FUNCTION_BLOCK Recipe_10054_Sixteen
VAR_INPUT
	execute: BOOL;
	Order: DUT_RECIPEORDER;
END_VAR
VAR_OUTPUT
	RecipeInfo: DUT_RECIPEOFFER;
	RecipeDone: BOOL;
	InitDone: BOOL;
	Ready: BOOL;
END_VAR
VAR
	userparametersum: LREAL;
	StepDone: BOOL;
	i: INT;
	Command: ARRAY[1..5] OF DUT_RecipeCommand;
	NextSkill: BOOL;
	SectionReady: BOOL;
END_VAR

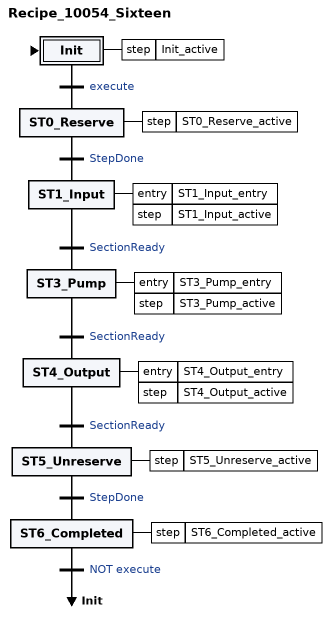
INITIAL_STEP Init:
    Init_active(N);  // step action
END_STEP
TRANSITION FROM Init TO ST0_Reserve
    := execute;
END_TRANSITION
STEP ST0_Reserve:
    ST0_Reserve_active(N);  // step action
END_STEP
TRANSITION FROM ST0_Reserve TO ST1_Input
    := StepDone;
END_TRANSITION
STEP ST1_Input:
    ST1_Input_entry(P1);  // entry action
    ST1_Input_active(N);  // step action
END_STEP
TRANSITION FROM ST1_Input TO ST3_Pump
    := SectionReady;
END_TRANSITION
STEP ST3_Pump:
    ST3_Pump_entry(P1);  // entry action
    ST3_Pump_active(N);  // step action
END_STEP
TRANSITION FROM ST3_Pump TO ST4_Output
    := SectionReady;
END_TRANSITION
STEP ST4_Output:
    ST4_Output_entry(P1);  // entry action
    ST4_Output_active(N);  // step action
END_STEP
TRANSITION FROM ST4_Output TO ST5_Unreserve
    := SectionReady;
END_TRANSITION
STEP ST5_Unreserve:
    ST5_Unreserve_active(N);  // step action
END_STEP
TRANSITION FROM ST5_Unreserve TO ST6_Completed
    := StepDone;
END_TRANSITION
STEP ST6_Completed:
    ST6_Completed_active(N);  // step action
END_STEP
TRANSITION FROM ST6_Completed TO Init
    := NOT execute;
END_TRANSITION

ACTION ST32b_Dose_exit:

END_ACTION

ACTION ST40_TransOutput_active:
//RT: 2014.11.23: Mover zum Output
StepDone := FALSE;

//Skill auswählen
ExecuteSkill.SkillID 		:= 1320;
ExecuteSkill.SkillName	 	:= 'Transport';

//Parameter setzen

ExecuteSkill.Parameter[3].ID := 3;
ExecuteSkill.Parameter[3].Name := 'Velocity';
ExecuteSkill.Parameter[3].Value := 300;



ExecuteSkill.Parameter[1].ID :=  1;
ExecuteSkill.Parameter[1].Name := 'TargetPosition X';
ExecuteSkill.Parameter[1].Value := 30 ;
ExecuteSkill.Parameter[1].StringValue := '#DP#2#XPosition';



ExecuteSkill.Parameter[2].ID := 2;
ExecuteSkill.Parameter[2].Name := 'TargetPosition Z';
ExecuteSkill.Parameter[2].Value := 100;// ZCookieModule - ZCookieModuleCalibration - 2* Cookiethickness + toppingthickness+ Preasureheight  ;



(* ExecuteSkill.Parameter[4].ID := 4;
ExecuteSkill.Parameter[4].Name := 'Acceleration';
ExecuteSkill.Parameter[4].Value :=0 ;

*)
(*
ExecuteSkill.Parameter[5].ID := ;
ExecuteSkill.Parameter[5].Name := '';
ExecuteSkill.Parameter[5].Value := ;
*)



ExecuteSkill();

StepDone := ExecuteSkill.Done;
END_ACTION

ACTION ST12_Input_active:
//RT: 2014.11.23: Input Modul auslösen
StepDone := FALSE;

//Skill auswählen
ExecuteSkill.SkillID 		:= 1402;
ExecuteSkill.SkillName	 	:= 'Input';

//Parameter setzen

ExecuteSkill.Parameter[1].ID := 1;
ExecuteSkill.Parameter[1].Name := 'TaskID';
ExecuteSkill.Parameter[1].Value := Order.TaskID;


(*
ExecuteSkill.Parameter[2].ID := ;
ExecuteSkill.Parameter[2].Name := '';
ExecuteSkill.Parameter[2].Value := ;
*)

(*
ExecuteSkill.Parameter[3].ID := ;
ExecuteSkill.Parameter[3].Name := '';
ExecuteSkill.Parameter[3].Value := ;
*)

(*
ExecuteSkill.Parameter[4].ID := ;
ExecuteSkill.Parameter[4].Name := '';
ExecuteSkill.Parameter[4].Value := ;
*)

(*
ExecuteSkill.Parameter[5].ID := ;
ExecuteSkill.Parameter[5].Name := '';
ExecuteSkill.Parameter[5].Value := ;
*)



ExecuteSkill();

StepDone := ExecuteSkill.Done;
END_ACTION

ACTION ST13_UnblockInput_active:
//RT: 2014.11.23: Gibt Mover Position Frei
StepDone := FALSE;

//Skill auswählen
ExecuteSkill.SkillID 		:= 1316;
ExecuteSkill.SkillName	 	:= 'Unblock';

//Parameter setzen

ExecuteSkill.Parameter[1].ID := 1;
ExecuteSkill.Parameter[1].Name := 'TaskID';
ExecuteSkill.Parameter[1].Value := Order.TaskID;


(*
ExecuteSkill.Parameter[2].ID := ;
ExecuteSkill.Parameter[2].Name := '';
ExecuteSkill.Parameter[2].Value := ;
*)

(*
ExecuteSkill.Parameter[3].ID := ;
ExecuteSkill.Parameter[3].Name := '';
ExecuteSkill.Parameter[3].Value := ;
*)

(*
ExecuteSkill.Parameter[4].ID := ;
ExecuteSkill.Parameter[4].Name := '';
ExecuteSkill.Parameter[4].Value := ;
*)

(*
ExecuteSkill.Parameter[5].ID := ;
ExecuteSkill.Parameter[5].Name := '';
ExecuteSkill.Parameter[5].Value := ;
*)



ExecuteSkill();

StepDone := ExecuteSkill.Done;
END_ACTION

ACTION ST42_CocktailOutput_active:
//RT: 2014.11.23: Ausgeben des Produktes
StepDone := FALSE;

//Skill auswählen
ExecuteSkill.SkillID 		:= 1403;
ExecuteSkill.SkillName	 	:= 'Output';

//Parameter setzen

ExecuteSkill.Parameter[1].ID := 1;
ExecuteSkill.Parameter[1].Name := 'TaskID';
ExecuteSkill.Parameter[1].Value := Order.TaskID;


(*
ExecuteSkill.Parameter[2].ID := ;
ExecuteSkill.Parameter[2].Name := '';
ExecuteSkill.Parameter[2].Value := ;
*)

(*
ExecuteSkill.Parameter[3].ID := ;
ExecuteSkill.Parameter[3].Name := '';
ExecuteSkill.Parameter[3].Value := ;
*)

(*
ExecuteSkill.Parameter[4].ID := ;
ExecuteSkill.Parameter[4].Name := '';
ExecuteSkill.Parameter[4].Value := ;
*)

(*
ExecuteSkill.Parameter[5].ID := ;
ExecuteSkill.Parameter[5].Name := '';
ExecuteSkill.Parameter[5].Value := ;
*)



ExecuteSkill();

StepDone := ExecuteSkill.Done;
END_ACTION

ACTION ST6_Completed_active:
//RT: 2014.11.23: Warte auf Execute = False
RecipeDone := TRUE;
StepDone := FALSE;
END_ACTION

ACTION ST4_Output_entry:
SectionReady := FALSE;
END_ACTION

ACTION ST44_Exit_active:
SectionReady := TRUE;
END_ACTION

ACTION ST4_Output_active:
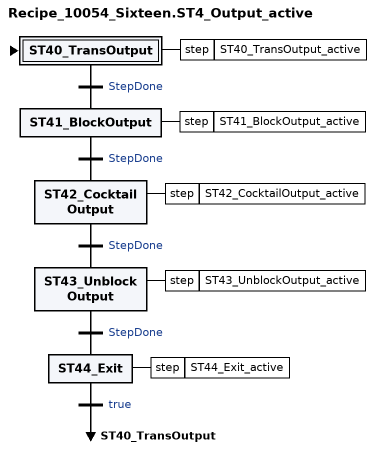
INITIAL_STEP ST40_TransOutput:
    ST40_TransOutput_active(N);  // step action
END_STEP
TRANSITION FROM ST40_TransOutput TO ST41_BlockOutput
    := StepDone;
END_TRANSITION
STEP ST41_BlockOutput:
    ST41_BlockOutput_active(N);  // step action
END_STEP
TRANSITION FROM ST41_BlockOutput TO ST42_CocktailOutput
    := StepDone;
END_TRANSITION
STEP ST42_CocktailOutput:
    ST42_CocktailOutput_active(N);  // step action
END_STEP
TRANSITION FROM ST42_CocktailOutput TO ST43_UnblockOutput
    := StepDone;
END_TRANSITION
STEP ST43_UnblockOutput:
    ST43_UnblockOutput_active(N);  // step action
END_STEP
TRANSITION FROM ST43_UnblockOutput TO ST44_Exit
    := StepDone;
END_TRANSITION
STEP ST44_Exit:
    ST44_Exit_active(N);  // step action
END_STEP
TRANSITION FROM ST44_Exit TO ST40_TransOutput
    := true;
END_TRANSITION
END_ACTION

ACTION Init_active:
//RT: 2014.11.23: Vorbereiten der daten und der HMI
RecipeDone := FALSE;

// Initialisation of Recipe Parameters an name etc
RecipeInfo.Name := 'Sixteen';
RecipeInfo.Description := '';
RecipeInfo.Dummy := FALSE;
RecipeInfo.RecipeID := 10054; 	// 
Initdone := TRUE;

//RT: 2014.11.23: wenn weniger als 5 alle lehren skills SkillID := 0
Command[1].SkillID := 1111;
Command[1].SkillName := 'Grenadine Syrup';
Command[1].Quantity := 11;

Command[2].SkillID := 1112;
Command[2].SkillName := 'Lemon Juice';
Command[2].Quantity := 11;

Command[3].SkillID := 1114;
Command[3].SkillName := 'Pineapple Juice';
Command[3].Quantity := 22;

Command[4].SkillID := 1117;
Command[4].SkillName := 'Orange Juice';
Command[4].Quantity := 45;

Command[5].SkillID := 1113;
Command[5].SkillName := 'Maracuja Juice';
Command[5].Quantity := 11;








//Parameter 0:

	RecipeInfo.UserParameter[0].Dummy 		:= FALSE;
	RecipeInfo.UserParameter[0].Default		:= 200;
	RecipeInfo.UserParameter[0].Description	:= 'Gives the total fluid amount in the glass';
	RecipeInfo.UserParameter[0].MaxValue	:= 200;
	RecipeInfo.UserParameter[0].MinValue	:= 10;
	RecipeInfo.UserParameter[0].Name		:= 'Total Liquid Amount';
	RecipeInfo.UserParameter[0].Unit		:= 'ml';
	
//Parameter 1-5:
FOR i := 1 TO 5 DO
	IF Command[i].SkillID = 0 THEN
		RecipeInfo.UserParameter[i].Dummy 		:= TRUE;
	ELSE
		RecipeInfo.UserParameter[i].Dummy 		:= FALSE;
		RecipeInfo.UserParameter[i].Default		:= Command[i].Quantity;
		RecipeInfo.UserParameter[i].Description	:= Command[i].SkillName;
		RecipeInfo.UserParameter[i].MaxValue	:= 100;
		RecipeInfo.UserParameter[i].MinValue	:= 1;
		RecipeInfo.UserParameter[i].Name		:= Command[i].SkillName;
		RecipeInfo.UserParameter[i].Unit		:= 'ml';	
	END_IF
END_FOR
END_ACTION

ACTION ST3_Pump_active:
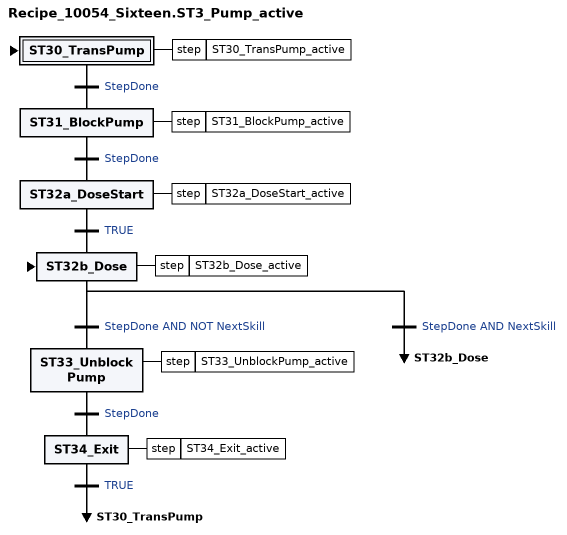
INITIAL_STEP ST30_TransPump:
    ST30_TransPump_active(N);  // step action
END_STEP
TRANSITION FROM ST30_TransPump TO ST31_BlockPump
    := StepDone;
END_TRANSITION
STEP ST31_BlockPump:
    ST31_BlockPump_active(N);  // step action
END_STEP
TRANSITION FROM ST31_BlockPump TO ST32a_DoseStart
    := StepDone;
END_TRANSITION
STEP ST32a_DoseStart:
    ST32a_DoseStart_active(N);  // step action
END_STEP
TRANSITION FROM ST32a_DoseStart TO ST32b_Dose
    := TRUE;
END_TRANSITION
STEP ST32b_Dose:
    ST32b_Dose_active(N);  // step action
END_STEP
TRANSITION FROM ST32b_Dose TO ST33_UnblockPump
    := StepDone AND NOT NextSkill;
END_TRANSITION
STEP ST33_UnblockPump:
    ST33_UnblockPump_active(N);  // step action
END_STEP
TRANSITION FROM ST33_UnblockPump TO ST34_Exit
    := StepDone;
END_TRANSITION
STEP ST34_Exit:
    ST34_Exit_active(N);  // step action
END_STEP
TRANSITION FROM ST34_Exit TO ST30_TransPump
    := TRUE;
END_TRANSITION
TRANSITION FROM ST32b_Dose TO ST32b_Dose
    := StepDone AND NextSkill;
END_TRANSITION
END_ACTION

ACTION ST34_Exit_active:
SectionReady := TRUE;
END_ACTION

ACTION ST10_TransToInput_active:
//RT: 2014.11.23: Mover zum Input

StepDone := FALSE;

//Skill auswählen
ExecuteSkill.SkillID 		:= 1320;
ExecuteSkill.SkillName	 	:= 'Transport';

//Parameter setzen

ExecuteSkill.Parameter[3].ID := 3;
ExecuteSkill.Parameter[3].Name := 'Velocity';
ExecuteSkill.Parameter[3].Value := 1000;



ExecuteSkill.Parameter[1].ID :=  1;
ExecuteSkill.Parameter[1].Name := 'TargetPosition X';
ExecuteSkill.Parameter[1].Value := 30 ;
ExecuteSkill.Parameter[1].StringValue := '#DP#2#XPosition';



ExecuteSkill.Parameter[2].ID := 2;
ExecuteSkill.Parameter[2].Name := 'TargetPosition Z';
ExecuteSkill.Parameter[2].Value := 100;// ZCookieModule - ZCookieModuleCalibration - 2* Cookiethickness + toppingthickness+ Preasureheight  ;



(*
ExecuteSkill.Parameter[4].ID := 4;
ExecuteSkill.Parameter[4].Name := 'Acceleration';
ExecuteSkill.Parameter[4].Value := 0 ;
*)

(*
ExecuteSkill.Parameter[5].ID := ;
ExecuteSkill.Parameter[5].Name := '';
ExecuteSkill.Parameter[5].Value := ;
*)



ExecuteSkill();

StepDone := ExecuteSkill.Done;
END_ACTION

ACTION ST1_Input_entry:
SectionReady := FALSE;
END_ACTION

ACTION ST32b_Dose_active:
//RT: 2014.11.23: Die Dosir Skills anlegen
StepDone := FALSE;

//Skill auswählen
ExecuteSkill.SkillID 		:= Command[i].SkillID;
ExecuteSkill.SkillName	 	:= Command[i].SkillName;
//Parameter setzen

ExecuteSkill.Parameter[0].ID := 1;
ExecuteSkill.Parameter[0].Name := 'Quantity';
//order.userParameter[0] = amount
ExecuteSkill.Parameter[0].Value := order.UserParameter[0].Value * order.UserParameter[i].Value / userparametersum ;//Summe aller Zutatenmengen;

(*
ExecuteSkill.Parameter[2].ID := ;
ExecuteSkill.Parameter[2].Name := '';
ExecuteSkill.Parameter[2].Value := ;
*)

(*
ExecuteSkill.Parameter[3].ID := ;
ExecuteSkill.Parameter[3].Name := '';
ExecuteSkill.Parameter[3].Value := ;
*)

(*
ExecuteSkill.Parameter[4].ID := ;
ExecuteSkill.Parameter[4].Name := '';
ExecuteSkill.Parameter[4].Value := ;
*)

(*
ExecuteSkill.Parameter[5].ID := ;
ExecuteSkill.Parameter[5].Name := '';
ExecuteSkill.Parameter[5].Value := ;
*)


ExecuteSkill();

StepDone := ExecuteSkill.Done;

i := i + 1 ;

IF i = 6 THEN
	NextSkill := FALSE;
ELSIF Command[i].SkillID = 0 THEN
	NextSkill := FALSE;
ELSE
	NextSkill := TRUE;
END_IF
END_ACTION

ACTION ST3_Pump_entry:
SectionReady := FALSE;
END_ACTION

ACTION ST43_UnblockOutput_active:
//RT: 2014.11.23: Gibt Mover Position Frei
StepDone := FALSE;

//Skill auswählen
ExecuteSkill.SkillID 		:= 1316;
ExecuteSkill.SkillName	 	:= 'Unblock';

//Parameter setzen

ExecuteSkill.Parameter[1].ID := 1;
ExecuteSkill.Parameter[1].Name := 'TaskID';
ExecuteSkill.Parameter[1].Value := Order.TaskID;


(*
ExecuteSkill.Parameter[2].ID := ;
ExecuteSkill.Parameter[2].Name := '';
ExecuteSkill.Parameter[2].Value := ;
*)

(*
ExecuteSkill.Parameter[3].ID := ;
ExecuteSkill.Parameter[3].Name := '';
ExecuteSkill.Parameter[3].Value := ;
*)

(*
ExecuteSkill.Parameter[4].ID := ;
ExecuteSkill.Parameter[4].Name := '';
ExecuteSkill.Parameter[4].Value := ;
*)

(*
ExecuteSkill.Parameter[5].ID := ;
ExecuteSkill.Parameter[5].Name := '';
ExecuteSkill.Parameter[5].Value := ;
*)



ExecuteSkill();

StepDone := ExecuteSkill.Done;
END_ACTION

ACTION ST1_Input_active:
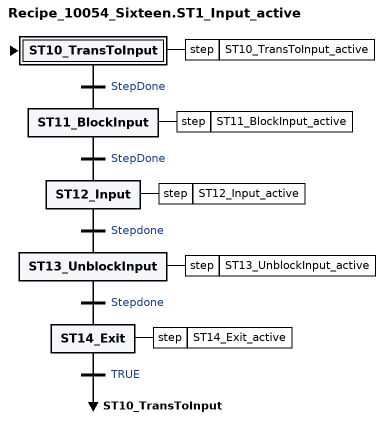
INITIAL_STEP ST10_TransToInput:
    ST10_TransToInput_active(N);  // step action
END_STEP
TRANSITION FROM ST10_TransToInput TO ST11_BlockInput
    := StepDone;
END_TRANSITION
STEP ST11_BlockInput:
    ST11_BlockInput_active(N);  // step action
END_STEP
TRANSITION FROM ST11_BlockInput TO ST12_Input
    := StepDone;
END_TRANSITION
STEP ST12_Input:
    ST12_Input_active(N);  // step action
END_STEP
TRANSITION FROM ST12_Input TO ST13_UnblockInput
    := Stepdone;
END_TRANSITION
STEP ST13_UnblockInput:
    ST13_UnblockInput_active(N);  // step action
END_STEP
TRANSITION FROM ST13_UnblockInput TO ST14_Exit
    := Stepdone;
END_TRANSITION
STEP ST14_Exit:
    ST14_Exit_active(N);  // step action
END_STEP
TRANSITION FROM ST14_Exit TO ST10_TransToInput
    := TRUE;
END_TRANSITION
END_ACTION

ACTION ST1_Reserve0_active:
//RT: 2014.11.23: Reservire einen Mover

StepDone := FALSE;
RecipeDone := FALSE;
//Skill auswählen
ExecuteSkill.SkillID 		:= 1310;
ExecuteSkill.SkillName	 	:= 'Reserve';

//Parameter setzen

ExecuteSkill.Parameter[1].ID := 1;
ExecuteSkill.Parameter[1].Name := 'TaskID';
ExecuteSkill.Parameter[1].Value := Order.TaskID;

(*
ExecuteSkill.Parameter[2].ID := ;
ExecuteSkill.Parameter[2].Name := '';
ExecuteSkill.Parameter[2].Value := ;
*)

(*
ExecuteSkill.Parameter[3].ID := ;
ExecuteSkill.Parameter[3].Name := '';
ExecuteSkill.Parameter[3].Value := ;
*)

(*
ExecuteSkill.Parameter[4].ID := ;
ExecuteSkill.Parameter[4].Name := '';
ExecuteSkill.Parameter[4].Value := ;
*)

(*
ExecuteSkill.Parameter[5].ID := ;
ExecuteSkill.Parameter[5].Name := '';
ExecuteSkill.Parameter[5].Value := ;
*)

ExecuteSkill();

StepDone := ExecuteSkill.Done;
END_ACTION

ACTION ST32a_DoseStart_active:
//RT: 2014.11.23: Summe aller zutaten zum Normiren

userparametersum := 0;
FOR i := 1 TO UserParameterCnt DO
	IF NOT (order.UserParameter[i].Value = 0) THEN
		userparametersum := userparametersum + order.UserParameter[i].Value;
	
	END_IF
END_FOR
IF userparametersum = 0 THEN
userparametersum := -1;
END_IF

//RT: 2014.11.23: Start wert des Arrays setzen
i := 1;
NextSkill := TRUE ;
END_ACTION

ACTION ST0_Reserve_active:
//RT: 2014.11.23: Reservire einen Mover

StepDone := FALSE;
RecipeDone := FALSE;
//Skill auswählen
ExecuteSkill.SkillID 		:= 1310;
ExecuteSkill.SkillName	 	:= 'Reserve';

//Parameter setzen

ExecuteSkill.Parameter[1].ID := 1;
ExecuteSkill.Parameter[1].Name := 'TaskID';
ExecuteSkill.Parameter[1].Value := Order.TaskID;

(*
ExecuteSkill.Parameter[2].ID := ;
ExecuteSkill.Parameter[2].Name := '';
ExecuteSkill.Parameter[2].Value := ;
*)

(*
ExecuteSkill.Parameter[3].ID := ;
ExecuteSkill.Parameter[3].Name := '';
ExecuteSkill.Parameter[3].Value := ;
*)

(*
ExecuteSkill.Parameter[4].ID := ;
ExecuteSkill.Parameter[4].Name := '';
ExecuteSkill.Parameter[4].Value := ;
*)

(*
ExecuteSkill.Parameter[5].ID := ;
ExecuteSkill.Parameter[5].Name := '';
ExecuteSkill.Parameter[5].Value := ;
*)

ExecuteSkill();

StepDone := ExecuteSkill.Done;
END_ACTION

ACTION ST5_Unreserve_active:
//RT: 2014.11.23: Mover Freigeben
StepDone := FALSE;

//Skill auswählen
ExecuteSkill.SkillID 		:= 1311;
ExecuteSkill.SkillName	 	:= 'Unreserve';

//Parameter setzen

ExecuteSkill.Parameter[1].ID := 1;
ExecuteSkill.Parameter[1].Name := 'TaskID';
ExecuteSkill.Parameter[1].Value := Order.TaskID;


(*
ExecuteSkill.Parameter[2].ID := ;
ExecuteSkill.Parameter[2].Name := '';
ExecuteSkill.Parameter[2].Val ue := ;
*)

(*
ExecuteSkill.Parameter[3].ID := ;
ExecuteSkill.Parameter[3].Name := '';
ExecuteSkill.Parameter[3].Value := ;
*)

(*
ExecuteSkill.Parameter[4].ID := ;
ExecuteSkill.Parameter[4].Name := '';
ExecuteSkill.Parameter[4].Value := ;
*)

(*
ExecuteSkill.Parameter[5].ID := ;
ExecuteSkill.Parameter[5].Name := '';
ExecuteSkill.Parameter[5].Value := ;
*)



ExecuteSkill();

StepDone := ExecuteSkill.Done;
END_ACTION

ACTION ST31_BlockPump_active:
//RT: 2014.11.23: Blockirt den Mover an Position
StepDone := FALSE;

//Skill auswählen
ExecuteSkill.SkillID 		:= 1315;
ExecuteSkill.SkillName	 	:= 'Block';

//Parameter setzen

ExecuteSkill.Parameter[1].ID := 1;
ExecuteSkill.Parameter[1].Name := 'TaskID';
ExecuteSkill.Parameter[1].Value := Order.TaskID;


(*
ExecuteSkill.Parameter[2].ID := ;
ExecuteSkill.Parameter[2].Name := '';
ExecuteSkill.Parameter[2].Value := ;
*)

(*
ExecuteSkill.Parameter[3].ID := ;
ExecuteSkill.Parameter[3].Name := '';
ExecuteSkill.Parameter[3].Value := ;
*)

(*
ExecuteSkill.Parameter[4].ID := ;
ExecuteSkill.Parameter[4].Name := '';
ExecuteSkill.Parameter[4].Value := ;
*)

(*
ExecuteSkill.Parameter[5].ID := ;
ExecuteSkill.Parameter[5].Name := '';
ExecuteSkill.Parameter[5].Value := ;
*)



ExecuteSkill();

StepDone := ExecuteSkill.Done;
END_ACTION

ACTION ST14_Exit_active:
SectionReady := TRUE;
END_ACTION

ACTION ST41_BlockOutput_active:
//RT: 2014.11.23: Blockirt den Mover an Position
StepDone := FALSE;

//Skill auswählen
ExecuteSkill.SkillID 		:= 1315;
ExecuteSkill.SkillName	 	:= 'Block';

//Parameter setzen

ExecuteSkill.Parameter[1].ID := 1;
ExecuteSkill.Parameter[1].Name := 'TaskID';
ExecuteSkill.Parameter[1].Value := Order.TaskID;


(*
ExecuteSkill.Parameter[2].ID := ;
ExecuteSkill.Parameter[2].Name := '';
ExecuteSkill.Parameter[2].Value := ;
*)

(*
ExecuteSkill.Parameter[3].ID := ;
ExecuteSkill.Parameter[3].Name := '';
ExecuteSkill.Parameter[3].Value := ;
*)

(*
ExecuteSkill.Parameter[4].ID := ;
ExecuteSkill.Parameter[4].Name := '';
ExecuteSkill.Parameter[4].Value := ;
*)

(*
ExecuteSkill.Parameter[5].ID := ;
ExecuteSkill.Parameter[5].Name := '';
ExecuteSkill.Parameter[5].Value := ;
*)



ExecuteSkill();

StepDone := ExecuteSkill.Done;
END_ACTION

ACTION ST33_UnblockPump_active:
//RT: 2014.11.23: Gibt Mover Position Frei
StepDone := FALSE;

//Skill auswählen
ExecuteSkill.SkillID 		:= 1316;
ExecuteSkill.SkillName	 	:= 'Unblock';

//Parameter setzen

ExecuteSkill.Parameter[1].ID := 1;
ExecuteSkill.Parameter[1].Name := 'TaskID';
ExecuteSkill.Parameter[1].Value := Order.TaskID;


(*
ExecuteSkill.Parameter[2].ID := ;
ExecuteSkill.Parameter[2].Name := '';
ExecuteSkill.Parameter[2].Value := ;
*)

(*
ExecuteSkill.Parameter[3].ID := ;
ExecuteSkill.Parameter[3].Name := '';
ExecuteSkill.Parameter[3].Value := ;
*)

(*
ExecuteSkill.Parameter[4].ID := ;
ExecuteSkill.Parameter[4].Name := '';
ExecuteSkill.Parameter[4].Value := ;
*)

(*
ExecuteSkill.Parameter[5].ID := ;
ExecuteSkill.Parameter[5].Name := '';
ExecuteSkill.Parameter[5].Value := ;
*)



ExecuteSkill();

StepDone := ExecuteSkill.Done;
END_ACTION

ACTION ST11_BlockInput_active:
//RT: 2014.11.23: Blockirt den Mover an Position
StepDone := FALSE;

//Skill auswählen
ExecuteSkill.SkillID 		:= 1315;
ExecuteSkill.SkillName	 	:= 'Block';

//Parameter setzen

ExecuteSkill.Parameter[1].ID := 1;
ExecuteSkill.Parameter[1].Name := 'TaskID';
ExecuteSkill.Parameter[1].Value := Order.TaskID;


(*
ExecuteSkill.Parameter[2].ID := ;
ExecuteSkill.Parameter[2].Name := '';
ExecuteSkill.Parameter[2].Value := ;
*)

(*
ExecuteSkill.Parameter[3].ID := ;
ExecuteSkill.Parameter[3].Name := '';
ExecuteSkill.Parameter[3].Value := ;
*)

(*
ExecuteSkill.Parameter[4].ID := ;
ExecuteSkill.Parameter[4].Name := '';
ExecuteSkill.Parameter[4].Value := ;
*)

(*
ExecuteSkill.Parameter[5].ID := ;
ExecuteSkill.Parameter[5].Name := '';
ExecuteSkill.Parameter[5].Value := ;
*)



ExecuteSkill();

StepDone := ExecuteSkill.Done;
END_ACTION

ACTION ST30_TransPump_active:
//RT: 2014.11.23: Mover zum Pump
StepDone := FALSE;

//Skill auswählen
ExecuteSkill.SkillID 		:= 1320;
ExecuteSkill.SkillName	 	:= 'Transport';

//Parameter setzen

ExecuteSkill.Parameter[3].ID := 3;
ExecuteSkill.Parameter[3].Name := 'Velocity';
ExecuteSkill.Parameter[3].Value := 1000;



ExecuteSkill.Parameter[1].ID :=  1;
ExecuteSkill.Parameter[1].Name := 'TargetPosition X';
ExecuteSkill.Parameter[1].Value := 30 ;
ExecuteSkill.Parameter[1].StringValue := '#DP#2#XPosition';



ExecuteSkill.Parameter[2].ID := 2;
ExecuteSkill.Parameter[2].Name := 'TargetPosition Z';
ExecuteSkill.Parameter[2].Value := 10;// ZCookieModule - ZCookieModuleCalibration - 2* Cookiethickness + toppingthickness+ Preasureheight  ;



(*
ExecuteSkill.Parameter[4].ID := 4;
ExecuteSkill.Parameter[4].Name := 'Acceleration';
ExecuteSkill.Parameter[4].Value := 0 ;
*)

(*
ExecuteSkill.Parameter[5].ID := ;
ExecuteSkill.Parameter[5].Name := '';
ExecuteSkill.Parameter[5].Value := ;
*)



ExecuteSkill();

StepDone := ExecuteSkill.Done;
END_ACTION

END_FUNCTION_BLOCK

(* stored: Version 1.1.0.1, ProductVersion 3.1.0.25
   POU Recipe_10054_Sixteen: Id {3d5a676f-07b0-4ca9-951c-b27f15c9d1cb}
   Action ST32b_Dose_exit: Id {034dfa98-bb01-40c3-8820-0e799336d0cb}
   Action ST40_TransOutput_active: Id {0d28497e-0ac9-43f7-9345-beb7d7d2e898}
   Action ST12_Input_active: Id {0e3c4375-1df1-4582-a7ca-3abc56d645f9}
   Action ST13_UnblockInput_active: Id {1529eaaf-f9e2-4101-851e-52894156acca}
   Action ST42_CocktailOutput_active: Id {1dec498a-fdab-4806-ac81-b31f8f20c30f}
   Action ST6_Completed_active: Id {254bcfbc-6a19-44f3-aea1-007465a3b7da}
   Action ST4_Output_entry: Id {330fab1a-de15-4e05-a1d5-b3fe6e256ddb}
   Action ST44_Exit_active: Id {4499ceae-c393-4760-bcef-19a756aae657}
   Action ST4_Output_active: Id {5c92a484-eebf-48f0-bc9b-6b9a2a01c02d}
   Action Init_active: Id {5d3c9318-eef9-48ad-9087-c064bec0c654}
   Action ST3_Pump_active: Id {5e2acf5b-d894-4e77-bc47-c25a4eb0273f}
   Action ST34_Exit_active: Id {643e7cc0-5f60-4e32-a6b2-23577258b390}
   Action ST10_TransToInput_active: Id {7afe027c-1c3d-4692-9d1d-1c9cc43cfcef}
   Action ST1_Input_entry: Id {7dc444a2-edd4-4c80-b0ba-28a5e7f879ee}
   Action ST32b_Dose_active: Id {86329684-68f4-4559-a0cb-338853f847a7}
   Action ST3_Pump_entry: Id {8fdaa715-4959-4876-9d80-df77346f08dd}
   Action ST43_UnblockOutput_active: Id {952c098d-c7b3-4145-8b9a-6e2482571d6c}
   Action ST1_Input_active: Id {97a91810-56fe-4d05-bb6f-0c047cf29c2c}
   Action ST1_Reserve0_active: Id {9cf81a8c-9c30-4407-b796-673cfdfc6ef8}
   Action ST32a_DoseStart_active: Id {b2636c03-1578-46da-8d00-efe4e8ae2497}
   Action ST0_Reserve_active: Id {bb2b48a1-6193-4514-8450-92761189c483}
   Action ST5_Unreserve_active: Id {bd2c637a-f95c-45b8-a0b7-e0e6eeab5a9b}
   Action ST31_BlockPump_active: Id {ca57052a-2832-4f46-b623-af520f0cda14}
   Action ST14_Exit_active: Id {d7d1a988-3c1d-47bc-996c-236f1f0a2142}
   Action ST41_BlockOutput_active: Id {e94e39f4-ba27-41f4-9d85-be05b955f967}
   Action ST33_UnblockPump_active: Id {ed4639a1-9b2a-41fe-bd79-3188a8eb9798}
   Action ST11_BlockInput_active: Id {efe4b08a-afd6-463a-9a4e-2d3216458164}
   Action ST30_TransPump_active: Id {fb915ec3-f7f1-4744-acf9-b9b1f86a73e2} *)
